Fanuc TP program (LS listing): h3_stop.ls

/PROG  H3_STOP
/ATTR
OWNER		= MNEDITOR;
COMMENT		= "";
PROG_SIZE	= 380;
CREATE		= DATE 19-04-11  TIME 16:02:20;
MODIFIED	= DATE 19-04-11  TIME 16:06:14;
FILE_NAME	= H2_STOP;
VERSION		= 0;
LINE_COUNT	= 14;
MEMORY_SIZE	= 860;
PROTECT		= READ_WRITE;
TCD:  STACK_SIZE	= 0,
      TASK_PRIORITY	= 50,
      TIME_SLICE	= 0,
      BUSY_LAMP_OFF	= 0,
      ABORT_REQUEST	= 0,
      PAUSE_REQUEST	= 0;
DEFAULT_GROUP	= 1,*,*,*,*;
CONTROL_CODE	= 00000000 00000000;
/APPL
/MN
   1:  DO[32]=PULSE,1.0sec ;
   2:  WAIT   1.00(sec) ;
   3:   ;
   4:  //$WAITTMOUT=200 ;
   5:  //WAIT (DI[48:W1_DOOR_CLOSED]) TIMEOUT,LBL[1] ;
   6:   ;
   7:   ;
   8:  END ;
   9:  LBL[1] ;
  10:  MESSAGE[...] ;
  11:  MESSAGE[VRATA STROJA 1] ;
  12:  MESSAGE[NISU ZATVORENA] ;
  13:  WAIT (DI[48:W1_DOOR_CLOSED])    ;
  14:  END ;
/POS
/END
